FUNCTION_BLOCK INTERNAL TestNode EXTENDS Node

METHOD PUBLIC Clone : I_Node
VAR_INPUT
END_VAR
END_METHOD

METHOD PROTECTED OnExecute : HRESULT
END_METHOD

METHOD SetId
VAR_INPUT
    Id : T_MaxString;
END_VAR
SUPER^._id := Id;
END_METHOD

END_FUNCTION_BLOCK

(* stored: Version 1.1.0.1, ProductVersion 3.1.4024.13
   POU TestNode: Id {742e5d1b-6d5a-0ae1-0d77-7a5b67fa5319}, SpecialFunc None
   Method Clone: Id {59346da4-47b6-0941-30c2-f0bc5cf38500}
   Method OnExecute: Id {d3f7e7fb-03f0-0202-1599-9d475e196221}
   Method SetId: Id {fe7e0319-7d10-0992-1191-1ae8bc11f3b4} *)
